INTERFACE ICommon

METHOD ConfigureRead : Block64Words
VAR_INPUT
END_VAR
//turns internal data(Retain arae , into 64Words block , pass to HMI
END_METHOD

METHOD ConfigureWrite : BOOL
VAR_INPUT
	input : Block64Words;
END_VAR
//turns 64Words blocki , into  nternal data(Retain arae, from HMI
END_METHOD

METHOD Control : BOOL
VAR_INPUT
	input : Block64Words;
END_VAR
END_METHOD

METHOD ErrorClear : BOOL
VAR_INPUT
	//reset,ignore
	input : eErrorClearWays;
END_VAR
END_METHOD

METHOD ErrorDetect : INT
VAR_INPUT
END_VAR
END_METHOD

METHOD Monitor : Block64Words
VAR_INPUT
END_VAR
END_METHOD

METHOD TypeCode : eTypeCodes
VAR_INPUT
END_VAR
END_METHOD

END_INTERFACE

(* stored: Version 1.1.0.1, ProductVersion 3.1.4022.10
   Itf ICommon: Id {3195de24-7332-4626-a0e0-5f82f7dad679}
   Method ConfigureRead: Id {6d589c03-f339-48ab-b876-cab398236125}
   Method ConfigureWrite: Id {632a7afa-57b4-410f-90c5-014e311845e0}
   Method Control: Id {bf54ab1c-a189-4b4e-a555-103d378be280}
   Method ErrorClear: Id {08c8aed5-bdc9-41ea-ada2-f017e55dd3f3}
   Method ErrorDetect: Id {ca40218d-104f-4911-94a5-fbf59c9d1e4d}
   Method Monitor: Id {b1eb2aa0-d7da-4a19-8768-e8a193343f37}
   Method TypeCode: Id {64ea1201-6b50-4ccb-bd12-8f3175ca76f8} *)
